{attribute 'linkalways'} 
{attribute 'no_explicit_call' := 'This FB is a CLASS and must be accessed using methods or properties'}
{attribute 'enable_dynamic_creation'}
FUNCTION_BLOCK _ETcVnCameraState EXTENDS EnumDatatypeBase
VAR
	localData : ETcVnCameraState;
	activeData : REFERENCE TO ETcVnCameraState;
	enumBaseDatatype : _DINT(localData);
END_VAR

METHOD PRIVATE AddLocalEnumeration
VAR_INPUT
	Enumeration : T_MAXSTRING;
	Value : ETcVnCameraState;
END_VAR
AddEnumeration(Enumeration, Value);
END_METHOD

PROPERTY PUBLIC Address : PVOID
GET
Address := ADR(activeData);
END_GET
END_PROPERTY

METHOD PUBLIC ClearReference
VAR_INPUT
END_VAR
activeData REF= localData;
SetBaseDatatypeReference();
END_METHOD

METHOD PUBLIC Clone : I_Datatype
VAR
    pClone : POINTER TO _ETcVnCameraState;
END_VAR
pClone := __NEW(_ETcVnCameraState(InitialValue := Value));
Clone := pClone^;
END_METHOD

METHOD FB_init : BOOL
VAR_INPUT
	bInitRetains : BOOL; // if TRUE, the retain variables are initialized (warm start / cold start)
	bInCopyCode : BOOL;  // if TRUE, the instance afterwards gets moved into the copy code (online change)
	InitialValue : ETcVnCameraState;
END_VAR
localData := InitialValue;
AddBaseDatatype(enumBaseDatatype);
ClearReference();

AddLocalEnumeration('TCVN_CS_ERROR', ETcVnCameraState.TCVN_CS_ERROR);
AddLocalEnumeration('TCVN_CS_INITIAL', ETcVnCameraState.TCVN_CS_INITIAL);
AddLocalEnumeration('TCVN_CS_INITIALIZING', ETcVnCameraState.TCVN_CS_INITIALIZING);
AddLocalEnumeration('TCVN_CS_INITIALIZED', ETcVnCameraState.TCVN_CS_INITIALIZED);
AddLocalEnumeration('TCVN_CS_OPENING', ETcVnCameraState.TCVN_CS_OPENING);
AddLocalEnumeration('TCVN_CS_OPENED', ETcVnCameraState.TCVN_CS_OPENED);
AddLocalEnumeration('TCVN_CS_STARTACQUISITION', ETcVnCameraState.TCVN_CS_STARTACQUISITION);
AddLocalEnumeration('TCVN_CS_ACQUIRING', ETcVnCameraState.TCVN_CS_ACQUIRING);
AddLocalEnumeration('TCVN_CS_STOPACQUISITION', ETcVnCameraState.TCVN_CS_STOPACQUISITION);
AddLocalEnumeration('TCVN_CS_RESETTINGFEATURES', ETcVnCameraState.TCVN_CS_RESETTINGFEATURES);
AddLocalEnumeration('TCVN_CS_TRIGGERING', ETcVnCameraState.TCVN_CS_TRIGGERING);
AddLocalEnumeration('TCVN_CS_CLOSING', ETcVnCameraState.TCVN_CS_CLOSING);
END_METHOD

PROPERTY PUBLIC Identifier : T_MAXSTRING
GET
Identifier := 'ETcVnCameraState';
END_GET
END_PROPERTY

METHOD IsEnumeratorValueEqual : BOOL
VAR_INPUT
	Enumerator : I_KeyValueForwardEnumerator;
END_VAR
VAR
	storedValue : ETcVnCameraState;
END_VAR
IF NOT Enumerator.TryGet(storedValue) THEN
	RETURN;
END_IF

IsEnumeratorValueEqual := storedValue = activeData;
END_METHOD

METHOD PUBLIC MakeReferenceTo
VAR_INPUT
	ReferenceTarget : REFERENCE TO ETcVnCameraState;
END_VAR
activeData REF= ReferenceTarget;
SetBaseDatatypeReference();
END_METHOD

METHOD PROTECTED SetBaseDatatypeReference
VAR_INPUT
END_VAR
enumBaseDatatype.MakeReferenceTo(activeData);
END_METHOD

PROPERTY PUBLIC Size : UDINT
GET
Size := SIZEOF(activeData);
END_GET
END_PROPERTY

METHOD TryMakeReferenceTo : BOOL
VAR_INPUT
	Target : I_Datatype;
END_VAR
VAR
	pTargetData : POINTER TO ETcVnCameraState;
END_VAR
IF NOT IsEquivalentTo(Target) THEN
	RETURN;
END_IF

pTargetData := Target.Address;
activeData REF= pTargetData^;
SetBaseDatatypeReference();
TryMakeReferenceTo := TRUE;
END_METHOD

PROPERTY PUBLIC Value : ETcVnCameraState
GET
Value := activeData;
END_GET
SET
activeData := Value;
END_SET
END_PROPERTY

END_FUNCTION_BLOCK

(* stored: Version 1.1.0.1, ProductVersion 3.1.4026.13
   POU _ETcVnCameraState: Id {45f1edd2-c105-4f78-971d-4b3f26100f3e}, SpecialFunc None
   Folder Core: Id {f4f85b97-5d80-0f3e-131b-ea19a41e3666}
   Folder Protected: Id {f6c103f3-e96b-08e4-127a-396c18be9062}
   Folder Customize: Id {4bb9b1bf-e4db-0bbf-1902-0fd0b27263f4}
   Folder Constructor: Id {e869d4ca-ff40-4dde-b922-3626e7b4258a}
   Folder Private: Id {6b7528fd-c49e-4520-a724-f1ab14d3528d}
   Folder Protected: Id {427cf71e-c2ec-4c86-a574-1c8a2c29ceba}
   Method AddLocalEnumeration: Id {51f265a2-95c2-4077-95c7-3d14ac35dda7}
   Property Address: Id {45435370-b1f6-0806-02e4-2f15a1e1776e}
   Get Get: Id {da524b49-e5ed-068a-19dd-e73ff6d5f5fa}
   Method ClearReference: Id {b62f62fa-2115-0c1c-3786-2d5755aa725e}
   Method Clone: Id {1d5432c0-33be-4703-8c3b-e24fe472799e}
   Method FB_init: Id {091616f5-73c1-45dd-9e61-d04f8ee45408}
   Property Identifier: Id {be4f896b-d3a3-408b-bdc8-de1062a0b3d4}
   Get Get: Id {9e164387-4d81-4bfe-99af-65dc246de864}
   Method IsEnumeratorValueEqual: Id {dfd7019f-075e-444b-8738-ffca7b01b69a}
   Method MakeReferenceTo: Id {575e687d-4a24-4411-bbd0-104a7abe0ce1}
   Method SetBaseDatatypeReference: Id {774a9970-95f9-03d1-17f0-06def55a232b}
   Property Size: Id {c094a220-bc50-032c-32b2-788387e2254b}
   Get Get: Id {5a3bd43f-5e0a-0794-24e6-7b4e55342dfa}
   Method TryMakeReferenceTo: Id {8d85677a-e761-4795-a160-4bfde707ac0b}
   Property Value: Id {c7b0bd3a-f90c-463c-a545-44949d16de32}
   Get Get: Id {4cf0a00c-7c38-4fef-8292-257a11790ca8}
   Set Set: Id {bfc722eb-b6ba-488c-831a-f3a688a8ac6c} *)
